TYPE ST_AlarmTimeInfos :
STRUCT
	Activated		: Tc2_Utilities.TIMESTRUCT;
	Deactivated		: Tc2_Utilities.TIMESTRUCT;
	Acknowledged	: Tc2_Utilities.TIMESTRUCT;
END_STRUCT
END_TYPE

(* stored: Version 1.1.0.1, ProductVersion 3.1.4024.13
   DUT ST_AlarmTimeInfos: Id {b07964f7-d2a7-0f87-180d-3ed0f874b372} *)
